(* CODESYS project Overzetter Simulatie Structured Tekst 2V0 - Leeg.project
   Company: Avans
   Description: Simulatie voor opstelling Sorteer Station.
   Title: Simulatie Sorteer Station
   Author: Rene Potters/Gerard Harkema
   Version: 0.1.0

Project tree, tasks and I/O mapping:
  Device : CODESYS Control Win V3, 3S - Smart Software Solutions GmbH, version 3.5.13.20
    application OverzetterSimulatie
      libraries: Standard, * (System); Util, * (System); VisuDialogs, 3.5.12.0 (System)
      task MainTask (cyclic, interval t#20ms, priority 1) calls Main
      task Simulatie (cyclic, interval t#20ms, priority 1) calls OverzetterSim
  Device_1 : EHV-CPU1025, Hitachi-IES, order no. EHV-CPU1025, version 3.5.4.11
      settings: IP Address = '192.168.1.31'
    application OverzetterRealWorld
      libraries: Standard, * (System); Util, * (System); VisuDialogs, 3.5.12.0 (System)
      task MainTask (cyclic, interval t#20ms, priority 1) calls Main
    Basic : Basic, Hitachi-IES, version 3.4.4.0
      <Empty>
      <Empty>
      <Empty>
      <Empty>
      <Empty>
      <Empty>
      <Empty>
      <Empty>
      <Empty>
      <Empty>
      <Empty>
  Simulatie/
    global variables SIM
    program OverzetterSim [ST]
    data type OverzetterDUT
  text list GlobalTextList
  Programma Structured Text/
    program Main [ST]
  global variables GVL
  Visualisaties/
    visualisation OverzetterHMI
*)

// Simulatie/OverzetterDUT
{attribute 'qualified_only'}
{attribute 'strict'}
TYPE OverzetterDUT :
(
	INHETMIDDEN, NAARRECHTS, ISRECHTS, NAARLINKS, ISLINKS, GEVALLEN
);
END_TYPE

// Simulatie/SIM
{attribute 'qualified_only'}
VAR_GLOBAL
	// Rotatie van de overzetter
	Vx_OvzRotate: INT := 0;
	// Visualisatie invisible blok
	Vx_OvzBlokLinks: BOOL := FALSE;
	// Visualisatie invisible blok
	Vx_OvzBlokOverzetter: BOOL := FALSE;
	// Visualisatie invisible blok
	Vx_OvzBlokRechts: BOOL := FALSE;
	// Visualisatie invisible blok
	Vx_OvzBlokGevallen: BOOL := FALSE;	
	// Magazijn opnieuw vullen (simulatie)
	Ix_MagazijnVullen 	: BOOL;
	// Goten legen (symulatie)
	Ix_GotenLegen	  	: BOOL;
	
	
	
	
	
	
	
	
	
	
	
	
	
	
	
	
	
	
	
	
	
	
	
	
	
	
	
	
	
	
	
	
	
	
	
	
	
	
	
	
	
	
	
	
	
	
	
	
	// Simulatie visualisatie 
	Vw_Rotate45: INT := 45;
	// Visualisatie X positie van de uitstoter
	Vw_MagUitstoterBekerX: INT := 30;
	// Visualisatie invisible blok uitgestoten
	Vx_MagBlokUit: BOOL := TRUE;
	// Visualisatie invisible blok 1
	Vx_MagBlok1: BOOL := TRUE;
	// Visualisatie invisible blok 2
	Vx_MagBlok2: BOOL := TRUE;
	// Visualisatie invisible blok 3
	Vx_MagBlok3: BOOL := TRUE;
	// Visualisatie invisible blok 4
	Vx_MagBlok4: BOOL := TRUE;
	// Visualisatie invisible blokken
	Vx_MagBlok: ARRAY[1..8] OF BOOL;
	// Aantal blokken in het magazijn
	Vw_MagBlokAantal: INT := 4;
	// Simulatie onthoudt dat een blok maar 1x wordt uitgestoten
	Vw_MagBlok1X: INT := 0;
	// Ligt er een blok op band
	Vw_SorBlokBand: BOOL := FALSE;
	// Rotatie van de stopper
	Vw_SorStopperRotate: INT := 0;
	// Rotatie van de stopper goot 1
	Vw_SorGoot1Rotate: INT := 0;
	// Rotatie van de stopper goot 2
	Vw_SorGoot2Rotate: INT := 0;
	// Kleur van de blok op betreffende positie
	Vw_SorKleurBand: DWORD := 0;
	// Bewegen van de blok over de band
	Vi_SorBlokBandX: INT := 0;
	// Bewegen van de blok over de band
	Vi_SorBlokBandY: INT := 0;
	// Simulatie error. Inverse logica.
	Vx_MagLuchtDrukError: BOOL := TRUE;
	// Simulatie error. Inverse logica.
	Vx_MagIsInError: BOOL := TRUE;
	// Simulatie error. Inverse logica.
	Vx_MagIsUitError: BOOL := TRUE;
	// Simulatie error. Inverse logica.
	Vx_OvzLuchtDrukError: BOOL := TRUE;
	// Simulatie error. Inverse logica.
	Vx_OvzIsLinksError: BOOL := TRUE;
	// Simulatie error. Inverse logica.
	Vx_OvzIsRechtsError: BOOL := TRUE;
	// Simulatie error. Inverse logica.
	Vx_OvzVacuumError: BOOL := TRUE;
	// Simulatie error. Inverse logica.
	Vx_SorMotorAfvoerError: BOOL := TRUE;
	// Simulatie error. Inverse logica.
	Vx_SorGoot1InError: BOOL := TRUE;
	// Simulatie error. Inverse logica.
	Vx_SorGoot1UitError: BOOL := TRUE;
	// Simulatie error. Inverse logica.
	Vx_SorInGootError: BOOL := TRUE;
	// Ligt er een blok op de betreffende positie
	Vx_SorBlokGoot: ARRAY [1..3,1..6] OF BOOL;
	// Kleur van de blok op betreffende positie
	Vw_SorKleurGoot: ARRAY [1..3,1..6] OF DWORD;
END_VAR

// GVL
VAR_GLOBAL
	// Indrukken resetknop 
	Ix_Resetknop: BOOL;
	// Keuzeknop staat op hand
	Ix_Hand: BOOL;
	// Keuzeknop staat op auto
	Ix_Auto: BOOL;
	// Indrukken noodstop
	Ix_Noodstop: BOOL;
	// Bekers magazijn zijn op
	Ix_MagazijnLeeg: BOOL;
	// Beker is uit dekselmagazijn gestoten
	Ix_UitstoterBekerIn: BOOL;
	// Uitstoter Beker haalt nieuwe beker op
	Ix_UitstoterBekerUit: BOOL;
	// Indrukken startknop
	Ix_Stopknop: BOOL := TRUE;
	// Indrukken stopknop
	Ix_Startknop: BOOL;	
	//Perslucht is aanwezig
	Ix_PersluchtAanwezig :BOOL;
	//Werkstuk door overzetter opgepakt
	Ix_VacuumAanwezig :BOOL;
	//Overzetter haalt beker op(linker pos.)
	Ix_OverzetterIsLinks :BOOL;
	//Overzetter plaatst beker op sorteerpositie
	Ix_OverzetterIsRechts :BOOL;
	//Beker aanwezig op detectiepositie
	Ix_BekerAanwezig :BOOL;
	//Beker is van aluminium
	Ix_BekerMetaal :BOOL;
	//Beker reflecteert en is dus niet zwart
	Ix_BekerReflecteerd :BOOL;
	//Product is naar een van de goten gegaan
	Ix_BekerInGoot :BOOL;
	//Pusher uitvoergoot 1 is in
	Ix_UitvoerGoot1IsIn :BOOL;
	//Pusher uitvoergoot 2 is in
	Ix_UitvoerGoot2IsIn :BOOL;
	//Beker afvoeren is bezig
	Ix_StationAfvoerVrij :BOOL;
	//Pusher uitvoergoot 1 is uit
	Ix_UitvoerGoot1IsUit :BOOL;
	//Pusher uitvoergoot 2 is uit
	Ix_UitvoerGoot2IsUit :BOOL;
	// Beker uit magazijn stoten
	Qx_BekerUitstoten: BOOL;	
	//Beker oppakken
	Qx_VacuumAan :BOOL;
	//Beker loslaten
	Qx_BekerLossen :BOOL;
	//Overzetter naar bekermagazijn
	Qx_OverzetterLinks :BOOL;
	//Overzetter naar sorteerpositie
	Qx_OverzetterRechts :BOOL;
	//Transportband aan
	Qx_MotorAfvoerAan :BOOL;
	//Pusher goot 1 uit
	Qx_UitvoerGoot1Uit :BOOL;
	//Pusher goot 2 uit
	Qx_UitvoerGoot2Uit :BOOL;
	//Beker stoppen op band voor detectie
	Qx_StopperUit :BOOL;
	//Uitsorteren is bezet
	Qx_StationBezet :BOOL;
	// Visualisatie invisible Gele vlak
	Qx_GeleLamp: BOOL;
	// Visualisatie invisible groene vlak
	Qx_GroeneLamp: BOOL;
	// Visualisatie invisible rode vlak
	Qx_RodeLamp: BOOL;
END_VAR

// Programma Structured Text/Main
PROGRAM Main
VAR
END_VAR

END_PROGRAM

// Simulatie/OverzetterSim
PROGRAM OverzetterSim
VAR
	// Timer om overzetten te vertragen
	Fb_Pulse: BLINK;
	// Timer om overzetten te vertragen
	Fb_Trigger: F_TRIG;
	// Eerste keer om visualisatie te updaten
	Mx_FirstTime: BOOL := TRUE;
	// Afhandeling van de overzetter
	Me_OvzState: OverzetterDUT := OVERZETTERDUT.INHETMIDDEN;	
	// Afhandeling van het blokje
	Me_BlokState: OverzetterDUT := OVERZETTERDUT.INHETMIDDEN;	
	// Duurt even voor het vacuum aanwezig is
	Mi_VacuumCntr: INT := 0;	
END_VAR
VAR CONSTANT


	// Inverse logica
	INVISABLE: BOOL := TRUE;
	// Inverse logica
	VISABLE: BOOL := FALSE;

END_VAR

// Initialisatie.

IF (Mx_FirstTime) THEN
	Me_OvzState := OVERZETTERDUT.INHETMIDDEN;
	Me_BlokState := OVERZETTERDUT.ISLINKS;
	
	Mi_VacuumCntr := 0;
	SIM.Vx_OvzRotate := 0;
	Mx_FirstTime := FALSE;
END_IF

//
// Afhandelen van de pulse events. Hierdoor loopt de simulatie los van de 
// TASK tijd.
//
Fb_Pulse(ENABLE:=TRUE,TIMELOW:=T#100MS, TIMEHIGH:=T#100MS);
Fb_Trigger(CLK:=Fb_Pulse.OUT);


//
// Only if no emergency active, start handling the simulation.
//
IF (GVL.Ix_Noodstop) THEN
	Mx_FirstTime := TRUE;	
	RETURN;
END_IF
	
//
// The pulse determines the speed of the cilinder to move in
// ore move out. The cilinder is only moved if the airpressure 
// is available.
//
IF (Fb_Trigger.Q AND SIM.Vx_OvzLuchtDrukError) THEN
	
	//
	// De status van de arm wordt los afgehandeld van het blokje. De beweging
	// van de arm staat hier namelijk helemaal los van.
	//
	
	CASE Me_OvzState OF
		
		OVERZETTERDUT.INHETMIDDEN:
			// 
			// De arm is in beweging naar links of naar rechts.
			// Indien de arm in de uiterste positie is wordt er van 
			// state gewisseld. Aangezien de arm in beweging is staan
			// de eindschakelaars uit.
			//
			
			IF (GVL.Qx_OverzetterLinks) THEN
				IF (SIM.Vx_OvzRotate > -90) THEN
					GVL.Ix_OverzetterIsLinks := FALSE;	
					GVL.Ix_OverzetterIsRechts := FALSE;			
					SIM.Vx_OvzRotate := SIM.Vx_OvzRotate - 10;
				ELSE
					Me_OvzState := OVERZETTERDUT.ISLINKS;			
				END_IF	
				
			END_IF
				 
			IF (GVL.Qx_OverzetterRechts) THEN
				IF (SIM.Vx_OvzRotate < 90) THEN
					GVL.Ix_OverzetterIsLinks := FALSE;	
					GVL.Ix_OverzetterIsRechts := FALSE;				
					SIM.Vx_OvzRotate := SIM.Vx_OvzRotate + 10;
				ELSE
					Me_OvzState := OVERZETTERDUT.ISRECHTS;				
				END_IF			
			END_IF
				
		OVERZETTERDUT.ISLINKS:
		    //
			// Arm staat in een uiterste stand. Eindschakelaar is ingeschakeld.
			// Zodra de arm weer wordt bewogen verandert de state.
			//
			
			GVL.Ix_OverzetterIsLinks := TRUE AND SIM.Vx_OvzIsLinksError;	

			IF (GVL.Qx_OverzetterRechts AND NOT GVL.Qx_OverzetterLinks) THEN
				GVL.Ix_OverzetterIsLinks := FALSE;				
				Me_OvzState := OVERZETTERDUT.INHETMIDDEN;		
			END_IF
			
		OVERZETTERDUT.ISRECHTS:
		    //
			// Arm staat in een uiterste stand. Eindschakelaar is ingeschakeld.
			// Zodra de arm weer wordt bewogen verandert de state.
			//
		
			GVL.Ix_OverzetterIsRechts := TRUE AND SIM.Vx_OvzIsRechtsError;	

			IF (GVL.Qx_OverzetterLinks AND NOT GVL.Qx_OverzetterRechts) THEN
				GVL.Ix_OverzetterIsRechts := FALSE;				
				Me_OvzState := OVERZETTERDUT.INHETMIDDEN;		
			END_IF			
			
		END_CASE

	END_IF	

	//
	// De status van het blokje hangt af van een aantal stuursignalen zoals waar
	// de arm zich bevindt, of er vacuum is en of er een beker lossen wordt gegeven.
	//
	
	CASE Me_BlokState OF
		OVERZETTERDUT.ISLINKS:
			//
			// Als de arm links is moet er eerste een vacuum opgebouwd worden alvorens het blokje 
			// opgepakt kan worden. Daarna verandert de state. 
			//
			
			SIM.Vx_OvzBlokGevallen 	 := INVISABLE;
			SIM.Vx_OvzBlokLinks 	 := VISABLE;
			SIM.Vx_OvzBlokOverzetter := INVISABLE;
			SIM.Vx_OvzBlokRechts 	 := INVISABLE;
			
			IF (GVL.Qx_VacuumAan AND SIM.Vx_OvzVacuumError AND GVL.Ix_OverzetterIsLinks) AND (NOT GVL.Qx_BekerLossen) THEN
				Mi_VacuumCntr := Mi_VacuumCntr + 1;
			END_IF
			
			IF (NOT GVL.Qx_VacuumAan AND SIM.Vx_OvzVacuumError) THEN
				Mi_VacuumCntr := 0;
			END_IF

			GVL.Ix_VacuumAanwezig := (Mi_VacuumCntr > 50);
	
			IF  ( GVL.Ix_VacuumAanwezig AND (Me_OvzState = OVERZETTERDUT.INHETMIDDEN)) THEN
				Me_BlokState := OVERZETTERDUT.INHETMIDDEN;
			END_IF
			
		OVERZETTERDUT.INHETMIDDEN:
			//
			// Het blokje is in beweging zolang er vacuum is. Als er geen vacuum meer is
			// valt het blokje... Indien de arm helemaal rechts is kan het blokje gelost 
			// worden. Dit moet met een Bekerlossen ondanks het feit dat er
			// geen vacuum meer is....
			//
			
			SIM.Vx_OvzBlokGevallen 	 := INVISABLE;
			SIM.Vx_OvzBlokLinks 	 := INVISABLE;
			SIM.Vx_OvzBlokOverzetter := VISABLE;
			SIM.Vx_OvzBlokRechts 	 := INVISABLE;

		 	IF (GVL.Ix_OverzetterIsRechts) AND (NOT GVL.Qx_VacuumAan) AND (GVL.Qx_BekerLossen) THEN
				GVL.Ix_VacuumAanwezig := FALSE;
				Me_BlokState := OVERZETTERDUT.ISRECHTS;		
				RETURN;		
			END_IF
			
			IF (NOT GVL.Ix_OverzetterIsRechts) AND (NOT GVL.Ix_OverzetterIsLinks) AND(NOT GVL.Qx_VacuumAan) THEN
				GVL.Ix_VacuumAanwezig := FALSE;
				Me_BlokState := OVERZETTERDUT.GEVALLEN;				
			END_IF

		OVERZETTERDUT.ISRECHTS:	
		    // 
			// Blokje is gelost. Nu is het wachten tot de overzetter terug naar links wordt gestuurd. Daarna verdwijnt
			// het blokje automatisch.
			//
			
			SIM.Vx_OvzBlokGevallen 	 := INVISABLE;
			SIM.Vx_OvzBlokLinks 	 := INVISABLE;
			SIM.Vx_OvzBlokOverzetter := INVISABLE;
			SIM.Vx_OvzBlokRechts 	 := VISABLE;
			
			IF (NOT GVL.Ix_OverzetterIsRechts) THEN
				Me_BlokState := OVERZETTERDUT.ISLINKS;					
			END_IF

		OVERZETTERDUT.GEVALLEN:
			//
			// Blokje is gevallen..... Situatie herstelt zich zodra de arm helemaal links staat.
			//
				
			SIM.Vx_OvzBlokGevallen 	 := VISABLE;
			SIM.Vx_OvzBlokLinks 	 := INVISABLE;
			SIM.Vx_OvzBlokOverzetter := INVISABLE;
			SIM.Vx_OvzBlokRechts 	 := INVISABLE;
			
			IF (GVL.Ix_OverzetterIsLinks) THEN
				Me_BlokState := OVERZETTERDUT.ISLINKS;					
			END_IF				
	END_CASE

END_PROGRAM

// Visualisaties/OverzetterHMI
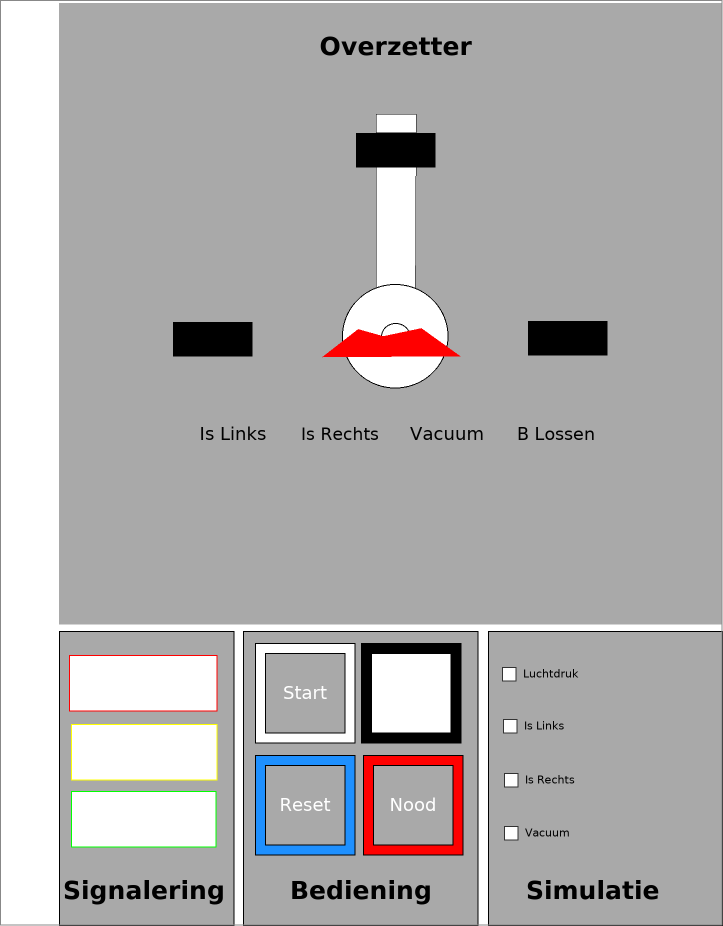
VISUALIZATION OverzetterHMI  // 723x926
    Rectangle (58,2 664x623)
    Polygon (233,394) (233,394) (273,434) (233,474) (193,434), "Is Links", colour toggle: Ix_OverzetterisLinks
    Polygon (340,394) (340,394) (380,434) (340,474) (300,434), "Is Rechts", colour toggle: Ix_OverzetterIsRechts
    Polygon (447,394) (447,394) (487,434) (447,474) (407,434), "Vacuum", colour toggle: Ix_VacuumAanwezig
    Polygon (376,131) (391,131) (416,131) (415,310) (376,310)
        p2858320360: SIM.Vx_OvzRotate
    Polygon (556,394) (556,394) (596,434) (556,474) (516,434), "B Lossen", colour toggle: Qx_BekerLossen
    Polygon (376,114) (391,114) (416,114) (416,132) (376,132), colour toggle: Qx_VacuumAan
        p2858320360: SIM.Vx_OvzRotate
    Polygon (356,133) (371,133) (435,133) (435,167) (356,167), invisible if: SIM.Vx_OvzBlokOverzetter
        p2277200375: SIM.Vx_OvzRotate
    Polygon (173,322) (188,322) (252,322) (252,356) (173,356), invisible if: SIM.Vx_OvzBlokLinks
    Polygon (528,321) (543,321) (607,321) (607,355) (528,355), invisible if: SIM.Vx_OvzBlokRechts
    Ellipse (342,284 106x104)
    Ellipse (381,323 29x27)
    Polygon (358,329) (383,336) (421,328) (460,356) (322,357), invisible if: SIM.Vx_OvzBlokGevallen
        p2277200375: SIM.Vx_OvzRotate
    Label (294,31 204x30), "Overzetter"
    Group (59,631 175x295)
        Rectangle (0,0 175x295)
        Rectangle (10,24 148x56), colour toggle: Qx_RodeLamp
        Rectangle (12,93 146x56), colour toggle: Qx_GeleLamp
        Rectangle (12,160 145x56), colour toggle: Qx_GroeneLamp
        Label (10,236 150x46), "Signalering"
    Group (243,631 235x295)
        Rectangle (0,0 235x295)
        Group (12,12 100x100)
            RoundedRectangle (0,0 100x100)
            RoundedRectangle (10,10 80x80), "Start", tooltip "Start knop", colour toggle: Ix_Startknop
                OnMouseDown: execute { Ix_Startknop := TRUE; }
                OnMouseUp: execute { Ix_Startknop := FALSE; }
        Group (118,12 100x100)
            RoundedRectangle (0,0 100x100)
            RoundedRectangle (10,10 80x80), "Stop", tooltip "Stop knop", colour toggle: Ix_Stopknop
                OnMouseDown: execute { Ix_Stopknop := FALSE; }
                OnMouseUp: execute { Ix_Stopknop := TRUE; }
        Group (12,124 100x100)
            RoundedRectangle (0,0 100x100)
            RoundedRectangle (10,10 80x80), "Reset", tooltip "Reset knop", colour toggle: Ix_Resetknop
                OnMouseDown: execute { Ix_Resetknop := TRUE; }
                OnMouseUp: execute { Ix_Resetknop := FALSE; }
        Group (120,124 100x100)
            RoundedRectangle (0,0 100x100), "Nood"
            RoundedRectangle (10,10 80x80), "Nood", tooltip "Noodstop", colour toggle: Ix_Noodstop
                OnMouseDown: execute { Ix_Noodstop := NOT Ix_Noodstop; }
        Label (43,236 150x46), "Bediening"
    Group (488,631 235x295)
        Group (0,0 235x295)
            Rectangle (0,0 235x295)
            Label (30,236 150x46), "Simulatie"
        Checkbox (12,17 196x52), "Luchtdruk", variable: SIM.Vx_OvzLuchtDrukError
        Checkbox (13,69 196x52), "Is Links", variable: SIM.Vx_OvzIsLinksError
        Checkbox (14,123 196x52), "Is Rechts", variable: SIM.Vx_OvzIsRechtsError
        Checkbox (14,176 196x52), "Vacuum", variable: SIM.Vx_OvzVacuumError
END_VISUALIZATION
